(* IEC 61131-3 sources: CS_4_Aufzugsteuerung/src/Stations/CP112/Steuerung/Class/clsCounter, 1 file *)

(* ---- clsCounter.st ---- *)
(*!
<Class
	Name               = "clsCounter"
	Revision           = "0.0"
	RealtimeTask       = "false"
	CyclicTask         = "false"
	BackgroundTask     = "false"
	Sigmatek           = "false"
	OSInterface        = "false"
	HighPriority       = "false"
	Automatic          = "false"
	UpdateMode         = "Prescan"
	SharedCommandTable = "true"
	Objectsize         = "(284,120)">
	<Channels>
		<Server Name="ClassSvr" Visualized="false" Initialize="false" WriteProtected="true" Retentive="false"/>
		<Server Name="Value" Visualized="false" Initialize="false" WriteProtected="true" Retentive="false"/>
	</Channels>
</Class>
*)
clsCounter : CLASS
  //Servers:
	ClassSvr 	: SvrChCmd_DINT;
	Value 	: SvrCh_DINT;
  //Clients:
  //Variables:
  //Functions:

	FUNCTION VIRTUAL GLOBAL CountUp;

	FUNCTION GLOBAL CountDown;

	FUNCTION GLOBAL Reset;
  //Tables:
	FUNCTION @STD
		VAR_OUTPUT
			ret_code	: CONFSTATES;
		END_VAR;
	FUNCTION GLOBAL TAB @CT_;
END_CLASS;

FUNCTION VIRTUAL GLOBAL clsCounter::CountUp
  Value += 1;
  Value.Write(input:=Value);
END_FUNCTION

FUNCTION GLOBAL clsCounter::CountDown
  Value -= 1;
END_FUNCTION

FUNCTION GLOBAL clsCounter::Reset
  Value := 0;
END_FUNCTION
